// TIA Portal V17 export
// export: Created 2024-09-02T12:50:25.3528773Z, ExportSetting WithDefaults, DisplayName Totally Integrated Automation Portal, DisplayVersion V17, DisplayName TIA Portal Openness, DisplayVersion V17, DisplayName TIA Portal Version Control Interface, DisplayVersion V17, DisplayName STEP 7 Professional, DisplayVersion V17, DisplayName STEP 7 Safety, DisplayVersion V17, DisplayName WinCC Professional, DisplayVersion V17
VAR_GLOBAL   // PLC tag table "GeneralSymbols"
   I_Circuit_breaker_24v_OK AT %I0.2 : Bool;   // Circuit breaker 24V DC IO (+S01-100FC3/-100FC6/-100FC8) / Leitungsschutzschalter 24V DC IO (+S01-100FC3/-100FC6/-100FC8)
   I_Circuit_breaker_230v_OK AT %I0.3 : Bool;   // Circuit breaker 230V DC IO (+S01-33FC01, 33FCB4, 33FB06/-44FC3/-44FC1) / Leitungsschutzschalter 230V AC IO (+S01-33FC01, 33FCB4, 33FB06/-44FC3/-44FC1)
   I_Circuit_breaker_400v_OK AT %I0.4 : Bool;   // Circuit breaker 400V DC IO (+S01-30QB7/-50QB8) / Leistungsschutzschalter 400V IO (+S01-30QB7/-50QB8)
   I_Scalance_OK AT %I0.5 : Bool;   // Scalance PN And ETH IO (+S01--275XF1) / Scalance PN und ETH IO (+S01-275XF1)
   I_Cabinet_temperatur_OK AT %I0.7 : Bool;   // Schaltschranktemperatur IO (+S01-- 300BT0.7)
   I_Controle_voltage_OK AT %I0.1 : Bool;   // Steuerspannung eingeschaltet (+S01-KF0)
   I_Safety_door_closed_OP70 AT %I1.2 : Bool;
   I_Safety_door_locked_OP70 AT %I1.3 : Bool;
   I_Button_Control_OFF AT %I2.1 : Bool;   // Taster NO Maschine aus (+ZP01-302SF2.1)
   I_Button_Control_ON AT %I2.0 : Bool;   // Taster NO Maschine ein (+ZP01-302SF2.0)
   I_Button_end_of_cycle_OP70 AT %I2.2 : Bool;   // Taster NO Halt bei Taktende (+ZP01-302SF2.2)
   I_Button_home_positioni_OP70 AT %I2.3 : Bool;   // Taster NO Grundstellungsfahrt (+ZP02-302SF2.4)
   I_Button_fault_ack_OP70 AT %I2.4 : Bool;   // Taster NO Störung Quittieren (+ZP01-302SF2.4)
   I_Vacuum_Gripper_Pressure_Ok AT %I3.0 : Bool;   // Taster NO Grundstellungsfahrt(+ZP01-302SF2.3)
   I_Feedback_circuit_enabling_safety AT %I3.4 : Bool;   // Rückführkreis Sicherheit Station
   I_Protective_door_OP70_K1 AT %I30.2 : Bool;   // Schutztür 1 Kanal 1 (+S01-SF30.2)
   I_Protective_door_OP70_K2 AT %I30.6 : Bool;   // Schutztür 1 Kanal 2 (+S01-SF30.6)
   "I_Safety_E-stop_OP70_K1" AT %I30.0 : Bool;   // Safety Not-Halt Kanal 1 (+ZP01-302SF30.0)
   "I_Safety_E-stop_OP70_K2" AT %I30.4 : Bool;   // Safety Not-Halt Kanal 2 (+ZP01-302SF30.4)
   Q_Control_voltage_ON AT %Q0.1 : Bool;   // Steuerspannung einschalten (+S01-600KF0.1)
   Q_Stop_at_cycle_end_OP70 AT %Q0.4 : Bool;   // Meldeleuchte Halt bei Taktende (+ZP01-600PF0.4)
   Q_Start_home_pos_OP70 AT %Q0.5 : Bool;   // Meldeleuchte Grundstellung Anfahren/Erreicht (+ZP01-600PF0.5)
   Q_warning_in_Station_OP70 AT %Q1.1 : Bool;   // Signalsäule Vorwarnung (+M01-611PF3.0)
   Q_fault_in_Station_OP70 AT %Q1.2 : Bool;   // Signalsäule Störung (+M01-611PF3.0)
   Q_Station_in_automatic_OP70 AT %Q1.0 : Bool;   // Signalsäule Verketter Betrieb(+M01-611PF3.0)
   Q_Protective_door_locking_OP70 AT %Q3.0 : Bool;
   Q_ScrewDriver_ON AT %Q2.4 : Bool;
   QF_Enable_Safety_Station AT %Q36.0 : Bool;
   Q_Air_Supply_Central_ON AT %Q50.1 : Bool;
   IEKS_OP70 AT %I7000.0 : "LTLL_typeEksInterface";   // EKS at the control panel / EKS am Bedienpult
   Q_Air_Supply_Vacumm_Gripper_ON AT %Q2.7 : Bool;
   Q_Door_Restart AT %Q3.3 : Bool;
END_VAR
